FUNCTION_BLOCK ASSEMBLE_AL_FROM_AD (* this Function combines the 2 AD (DWORD) adapters to a AL (LWORD) *)
  (* Standard: 61499-2; Description: Copyright (c) 2026 Meisterschulen am Ostbahnhof SPDX-License-Identifier: EPL-2.0 *)
  (* Version 1.0, 2026-05-16, Franz Höpfinger, Meisterschulen am Ostbahnhof, initial API and implementation and/or initial documentation *)
  PACKAGE adapter::assembling;
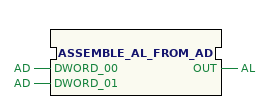
  SOCKETS
    DWORD_00 : adapter::types::unidirectional::AD; (* DWord 0 *)
    DWORD_01 : adapter::types::unidirectional::AD; (* DWord 1 *)
  END_SOCKETS
  PLUGS
    OUT : adapter::types::unidirectional::AL; (* LWORD Output *)
  END_PLUGS
END_FUNCTION_BLOCK
